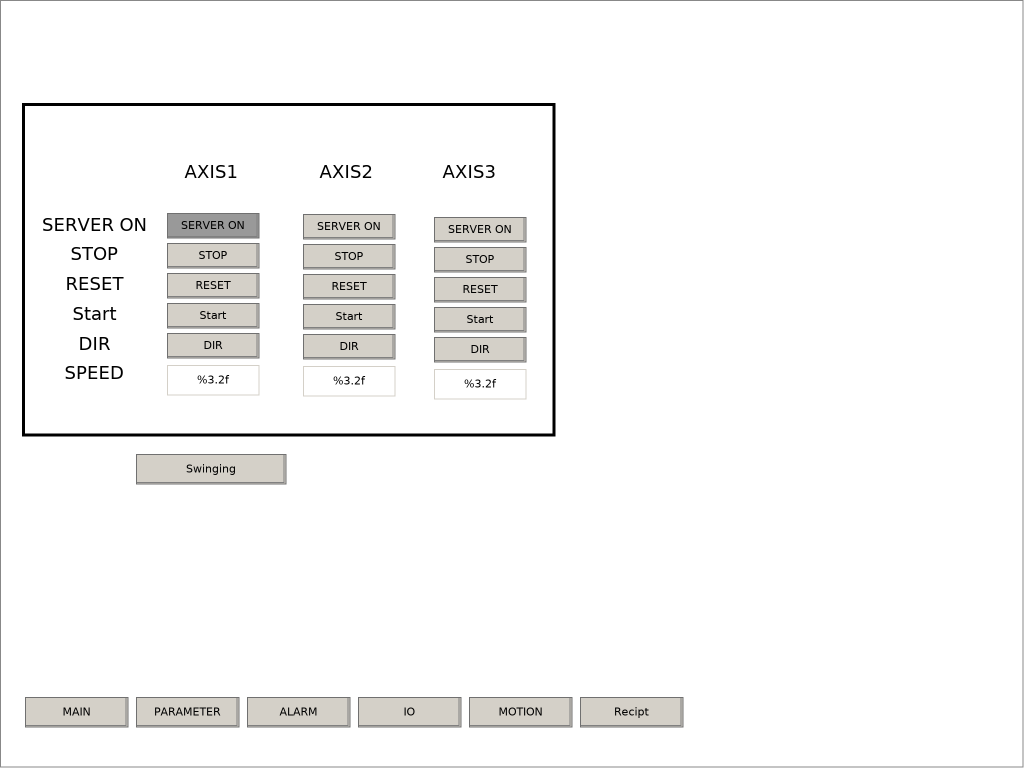
VISUALIZATION MOTION  // 1024x768, background image ImagePool_Base.base
    RoundedRectangle (22,103 533x333)
    Label (14,210 161x30), "SERVER ON"
    Label (14,239 161x30), "STOP"
    Label (14,269 161x30), "RESET"
    Label (14,299 161x30), "Start"
    Label (14,358 161x30), "SPEED"
    Button (167,213 92x25), "SERVER ON"
        toggle MOTION.Pwr_En_1 p2164770859=TRUE
    Button (167,243 92x25), "STOP"
        tap MOTION.stop_1
    Button (167,273 92x25), "RESET"
        tap MOTION.reset_1
    Button (167,303 92x25), "Start"
        tap MOTION.V_ex1
    Textfield (167,365 92x30), "%3.2f", text variable: MOTION.VV1
        OnMouseClick: write the text variable via Default, min 0, max 300
    Button (167,333 92x25), "DIR"
        toggle MOTION.DIR1
    Label (14,329 161x30), "DIR"
    Button (303,214 92x25), "SERVER ON"
        toggle MOTION.Pwr_En_2
    Button (303,244 92x25), "STOP"
        tap MOTION.stop_2
    Button (303,274 92x25), "RESET"
        tap MOTION.reset_2
    Button (303,304 92x25), "Start"
        tap MOTION.V_ex2
    Textfield (303,366 92x30), "%3.2f", text variable: MOTION.VV2
        OnMouseClick: write the text variable via Default, min 0, max 300
    Button (303,334 92x25), "DIR"
        toggle MOTION.DIR2
    Button (434,217 92x25), "SERVER ON"
        toggle MOTION.Pwr_En_3
    Button (434,247 92x25), "STOP"
        tap MOTION.stop_3
    Button (434,277 92x25), "RESET"
        tap MOTION.reset_3
    Button (434,307 92x25), "Start"
        tap MOTION.V_ex3
    Textfield (434,369 92x30), "%3.2f", text variable: MOTION.VV3
        OnMouseClick: write the text variable via Default, min 0, max 300
    Button (434,337 92x25), "DIR"
        toggle MOTION.DIR3 p2164770859=TRUE
    Label (155,157 113x30), "AXIS1"
    Label (290,157 113x30), "AXIS2"
    Label (413,157 113x30), "AXIS3"
    Button (136,454 150x30), "Swinging"
        toggle MOTION.swinging
    Button (25,697 103x30), "MAIN"
        OnMouseClick: change screen: MainBase
    Button (136,697 103x30), "PARAMETER"
        OnMouseClick: change screen: PARAMETER
    Button (247,697 103x30), "ALARM"
        OnMouseClick: change screen: ALARM
    Button (358,697 103x30), "IO"
        OnMouseClick: change screen: IO_TABLE
    Button (469,697 103x30), "MOTION"
        OnMouseClick: change screen: MOTION
    Button (580,697 103x30), "Recipt"
        OnMouseClick: change screen: Recipt
END_VISUALIZATION

(* stored: Version 1.1.0.1, ProductVersion 3.1.4024.11
   Visu MOTION: Id {642a5e26-6346-47ae-8a40-5c2188e9d1af} *)
